// SIMATIC S7-200 project (STEP 7-Micro/WIN), CPU 224 REL 02.01

SYMBOL_TABLE USER1
S0               I0.0     // EMERGENCY pushbutton for the control unit
S1               I0.1     // START green pushbutton for the control unit
S2               I0.2     // STOP red pushbutton for the control unit
S3               I0.3     // START green pushbutton for the control unit
S4               I0.4     // STOP red pushbutton for the control unit
S5               I0.5     // Inductive sensor for the conveyor unit 2
S6               I0.6     // Capacitive sensor for the conveyor unit 2
S11              I1.1     // Capacitive sensor for the conveyor unit 1
S12              I1.2     // REED limit switch for the conveyor unit 1
S13              I1.3     // REED limit switch for the conveyor unit 1
S14              I1.4     // REED limit switch for the conveyor unit 1
S3_OFF           M0.0     // Memory to turn off latch attached to S3
SS3              M0.1     // Output for latch attached to S3
R_T1             M0.2     // Internal relay to reset TIMER1
ALL_LAMP         M0.3     // Output to flash lamps H1, H2, H3 and H4
GREEN            M0.4     // Output to turn H1 and H3 permanently on for start run
S1_OFF           M0.5     // Memory to turn off latch attached to S1
SS1              M0.6     // Output for latch attached to S1
STOP_K2          M0.7     // Contact to stop K2 when piece is detected after 2 seconds
S13_OFF          M1.0     // Memory to turn off latch attached to S13
SS13_K1          M1.1     // Output for latch attached to S13 to start motor K1
SS13_K2          M1.2     // Output to start motor K2 when the pick and place unit is returning
SS5              M1.3     // Output for latch S6 the capacitive sensor
SS6              M1.4     // Output for latch S6 the capacitive sensor
C_STOP_K1        M1.5     // Stop conveyor belt 2 some time after capacitive piece is sensed
I_STOP_K1        M1.6     // Stop conveyor belt 2 some time after inductive piece is sensed
E_STOP           M1.7     // Activates EMERGENCY situation
S_STOP           M2.0     // Activates STOP situation
SS11             M2.1     // Latch for S11
S_STOP_OFF       M2.2     // Exit STOP Situation
E_STOP_OFF       M2.3     // Exit EMERGENCY Situation
RED              M2.4     // Output to stop flashing in emergency situation
S_H4             M2.5     // Output for lamp H4 in stop situation
Y8               Q0.0     // Solenoid valve for vacuum unit
H1               Q0.1     // Green Lamp pushbutton for the control unit
H2               Q0.2     // Red Lamp pushbutton for the control unit
H3               Q0.3     // Green Lamp pushbutton for the control unit
H4               Q0.4     // Red lamp pushbutton for the control unit
K1               Q1.0     // AC 1 phase motor relay for the conveyor unit 2
K2               Q1.1     // AC 1 phase motor relay for the conveyor unit 1
Y2               Q2.2     // Pushing cylinder solenoid valve for inuductive pieces
Y3               Q2.3     // Pushing cylinder solenoid valve for capacitive pieces
Y4               Q2.4     // Solenoid valve for magazine pieces pushing cylinder conveyor unit 1
Y5               Q2.5     // Solenoid valve for transport cylinder delivery conveyor unit 1
Y6               Q2.6     // Solenoid valve for transport cylinder return conveyour unit 1
Y7               Q2.7     // Solenoid valve for vacuum unit lifting cylinder conveyour unit 1
TIMER1           T37      // TON timer to flash all the lights
TIMER2           T38      // TON timer to check if piece is detected by S11
TIMER3           T39      // TON timer for events after a piece has been detected
TIMER4           T41      // TON timer started by inductive load being sensed
TIMER5           T42      // TON timer started by capacitive load being sensed
END_SYMBOL_TABLE

ORGANIZATION_BLOCK MAIN:OB1
TITLE=PROGRAM COMMENTS
BEGIN
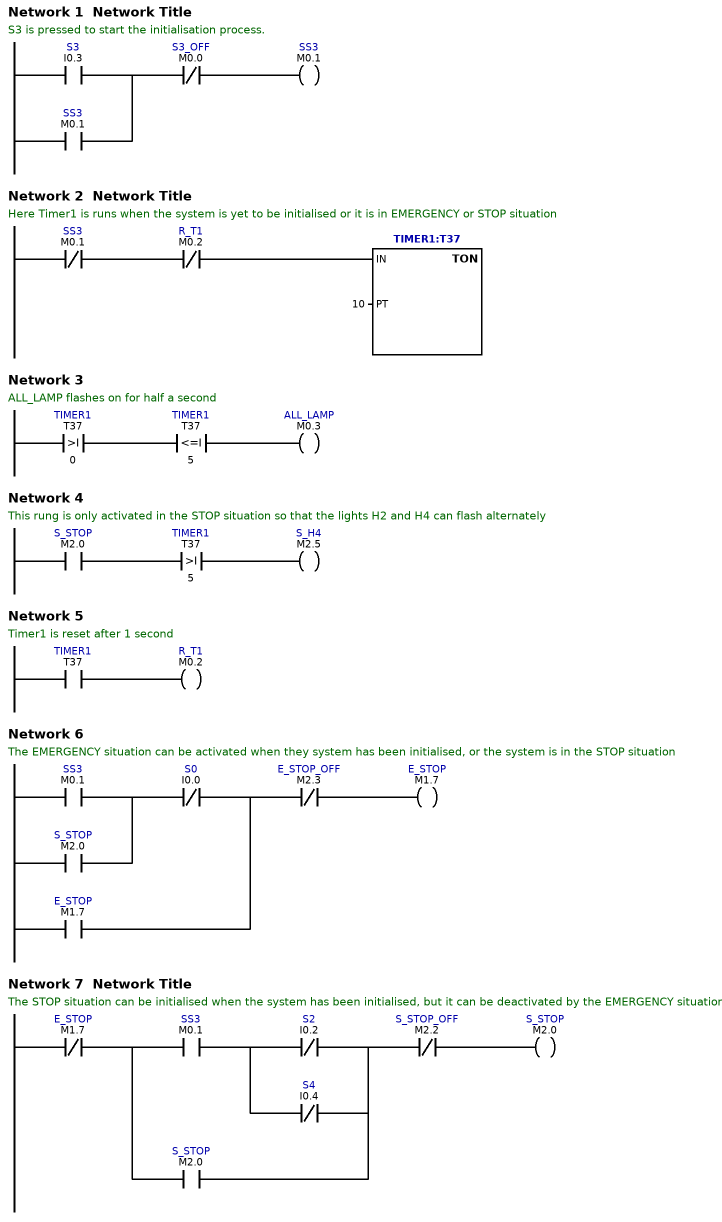
Network 1 // Network Title
// S3 is pressed to start the initialisation process.
LD     S3:I0.3
O      SS3:M0.1
AN     S3_OFF:M0.0
=      SS3:M0.1
Network 2 // Network Title
// Here Timer1 is runs when the system is yet to be initialised or it is in EMERGENCY or STOP situation
LDN    SS3:M0.1
AN     R_T1:M0.2
TON    TIMER1:T37, 10
Network 3
// ALL_LAMP flashes on for half a second
LDW>   TIMER1:T37, 0
AW<=   TIMER1:T37, 5
=      ALL_LAMP:M0.3
Network 4
// This rung is only activated in the STOP situation so that the lights H2 and H4 can flash alternately
// (network saved uncompiled; LAD cells follow)
// row 0: c0 -| |- S_STOP:M2.0  c1 -|>I|- TIMER1:T37, 5  c2 -( ) S_H4:M2.5
Network 5
// Timer1 is reset after 1 second
LD     TIMER1:T37
=      R_T1:M0.2
Network 6
// The EMERGENCY situation can be activated when they system has been initialised, or the system is in the STOP situation
// (network saved uncompiled; LAD cells follow)
// row 0: c0 -| |- SS3:M0.1 v  c1 -|/|- S0:I0.0 v  c2 -|/|- E_STOP_OFF:M2.3  c3 -( ) E_STOP:M1.7
// row 1: c0 -| |- S_STOP:M2.0 ^  c1 ^v
// row 2: c0 -| |- E_STOP:M1.7  c1 -- ^
Network 7 // Network Title
// The STOP situation can be initialised when the system has been initialised, but it can be deactivated by the EMERGENCY situation.
// (network saved uncompiled; LAD cells follow)
// row 0: c0 -|/|- E_STOP:M1.7 v  c1 -| |- SS3:M0.1 v  c2 -|/|- S2:I0.2 v  c3 -|/|- S_STOP_OFF:M2.2  c4 -( ) S_STOP:M2.0
// row 1: c0 ^v  c1 ^  c2 -|/|- S4:I0.4 ^v
// row 2: c0 ^  c1 -| |- S_STOP:M2.0  c2 -- ^
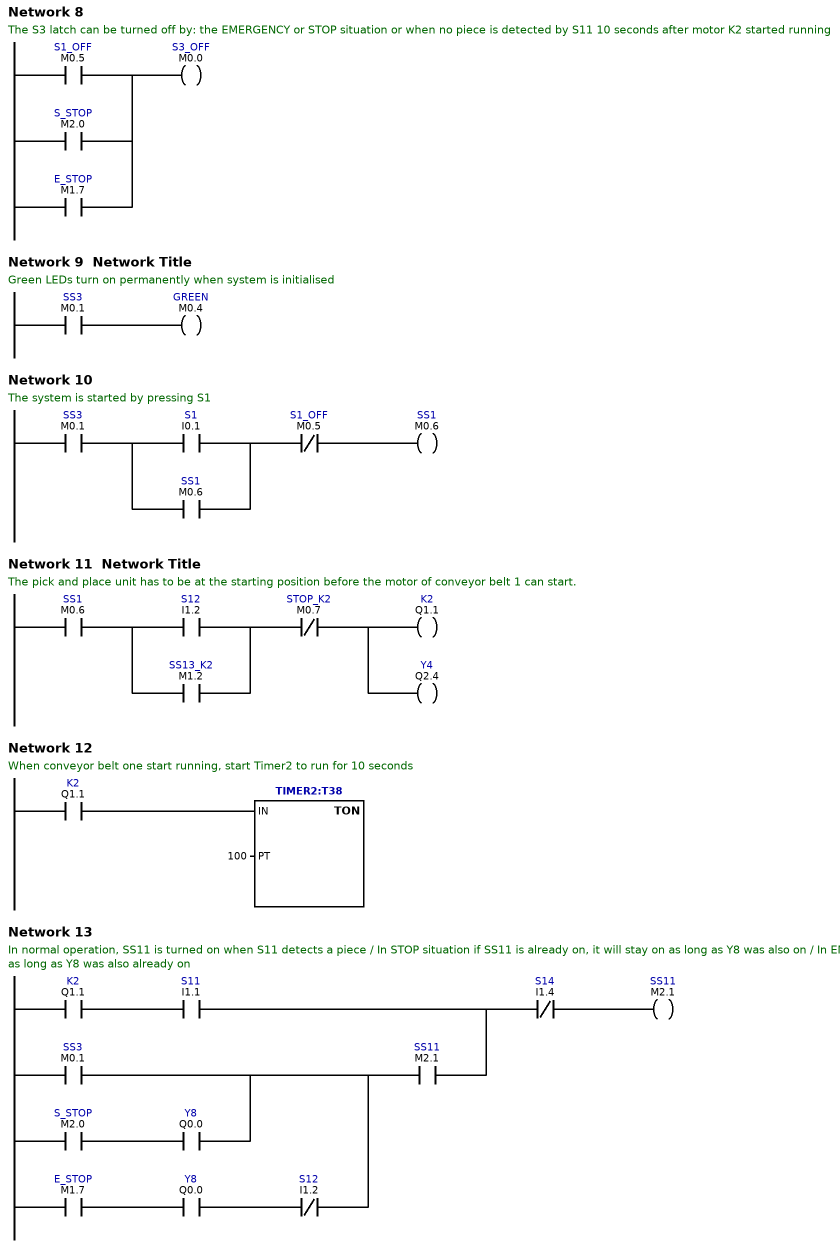
Network 8
// The S3 latch can be turned off by: the EMERGENCY or STOP situation or when no piece is detected by S11 10 seconds after motor K2 started running
// (network saved uncompiled; LAD cells follow)
// row 0: c0 -| |- S1_OFF:M0.5 v  c1 -( ) S3_OFF:M0.0
// row 1: c0 -| |- S_STOP:M2.0 ^v
// row 2: c0 -| |- E_STOP:M1.7 ^
Network 9 // Network Title
// Green LEDs turn on permanently when system is initialised
LD     SS3:M0.1
=      GREEN:M0.4
Network 10
// The system is started by pressing S1
LD     SS3:M0.1
LD     S1:I0.1
O      SS1:M0.6
ALD
AN     S1_OFF:M0.5
=      SS1:M0.6
Network 11 // Network Title
// The pick and place unit has to be at the starting position before the motor of conveyor belt 1 can start.
// (network saved uncompiled; LAD cells follow)
// row 0: c0 -| |- SS1:M0.6 v  c1 -| |- S12:I1.2 v  c2 -|/|- STOP_K2:M0.7 v  c3 -( ) K2:Q1.1
// row 1: c0 ^  c1 -| |- SS13_K2:M1.2 ^  c2 ^  c3 -( ) Y4:Q2.4
Network 12
// When conveyor belt one start running, start Timer2 to run for 10 seconds
LD     K2:Q1.1
TON    TIMER2:T38, 100
Network 13
// In normal operation, SS11 is turned on when S11 detects a piece
// In STOP situation if SS11 is already on, it will stay on as long as Y8 was also on
// In EMERGENCY if SS11 is already on, it will stay on as long as Y8 was also already on
// (network saved uncompiled; LAD cells follow)
// row 0: c0 -| |- K2:Q1.1  c1 -| |- S11:I1.1  c2 --  c3 -- v  c4 -|/|- S14:I1.4  c5 -( ) SS11:M2.1
// row 1: c0 -| |- SS3:M0.1  c1 -- v  c2 -- v  c3 -| |- SS11:M2.1 ^
// row 2: c0 -| |- S_STOP:M2.0  c1 -| |- Y8:Q0.0 ^  c2 ^v
// row 3: c0 -| |- E_STOP:M1.7  c1 -| |- Y8:Q0.0  c2 -|/|- S12:I1.2 ^
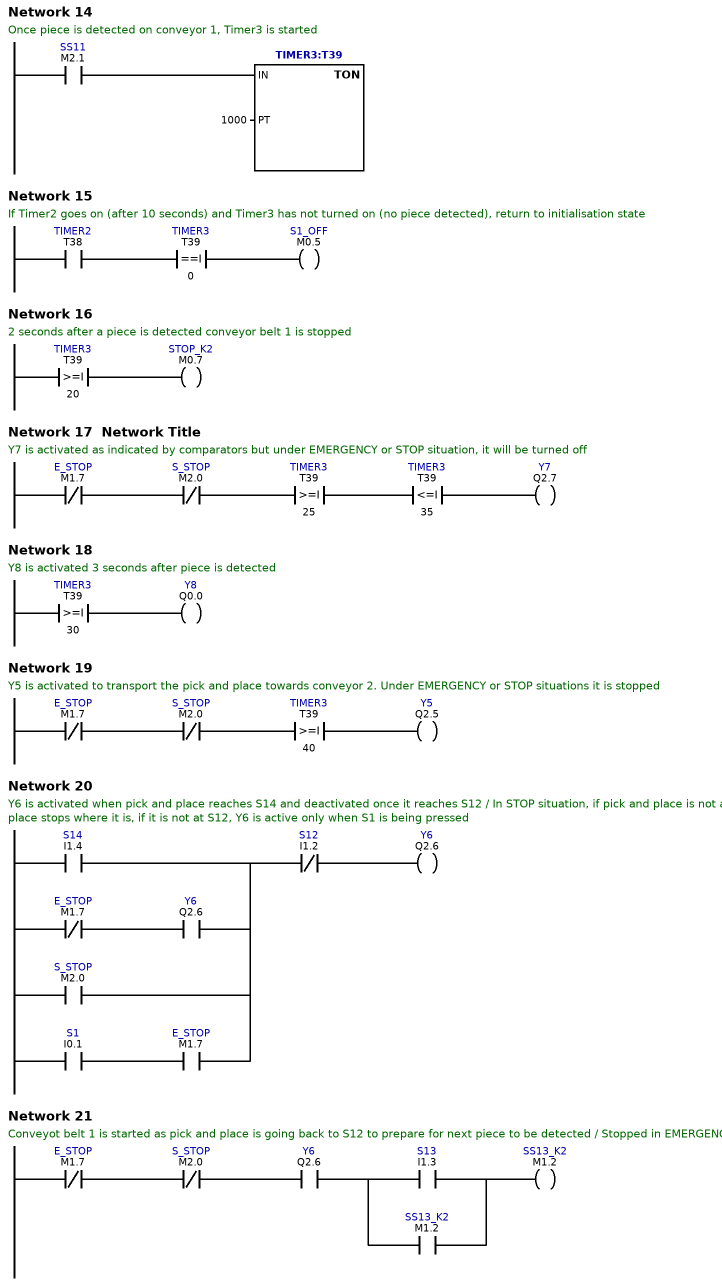
Network 14
// Once piece is detected on conveyor 1, Timer3 is started
// (network saved uncompiled; LAD cells follow)
// row 0: c0 -| |- SS11:M2.1  c1 --  c2 [TON TIMER3:T39 IN:=power@row0, PT:=1000]
// row 1: c2 [box]
Network 15
// If Timer2 goes on (after 10 seconds) and Timer3 has not turned on (no piece detected), return to initialisation state
LD     TIMER2:T38
AW=    TIMER3:T39, 0
=      S1_OFF:M0.5
Network 16
// 2 seconds after a piece is detected conveyor belt 1 is stopped
LDW>=  TIMER3:T39, 20
=      STOP_K2:M0.7
Network 17 // Network Title
// Y7 is activated as indicated by comparators but under EMERGENCY or STOP situation, it will be turned off
// (network saved uncompiled; LAD cells follow)
// row 0: c0 -|/|- E_STOP:M1.7  c1 -|/|- S_STOP:M2.0  c2 -|>=I|- TIMER3:T39, 25  c3 -|<=I|- TIMER3:T39, 35  c4 -( ) Y7:Q2.7
Network 18
// Y8 is activated 3 seconds after piece is detected
LDW>=  TIMER3:T39, 30
=      Y8:Q0.0
Network 19
// Y5 is activated to transport the pick and place towards conveyor 2. Under EMERGENCY or STOP situations it is stopped
// (network saved uncompiled; LAD cells follow)
// row 0: c0 -|/|- E_STOP:M1.7  c1 -|/|- S_STOP:M2.0  c2 -|>=I|- TIMER3:T39, 40  c3 -( ) Y5:Q2.5
Network 20
// Y6 is activated when pick and place reaches S14 and deactivated once it reaches S12
// In STOP situation, if pick and place is not at S12, Y6 is activated to return it
// In EMERGENCY situation, pick and place stops where it is, if it is not at S12, Y6 is active only when S1 is being pressed
// (network saved uncompiled; LAD cells follow)
// row 0: c0 -| |- S14:I1.4  c1 -- v  c2 -|/|- S12:I1.2  c3 -( ) Y6:Q2.6
// row 1: c0 -|/|- E_STOP:M1.7  c1 -| |- Y6:Q2.6 ^v
// row 2: c0 -| |- S_STOP:M2.0  c1 -- ^v
// row 3: c0 -| |- S1:I0.1  c1 -| |- E_STOP:M1.7 ^
Network 21
// Conveyot belt 1 is started as pick and place is going back to S12 to prepare for next piece to be detected
// Stopped in EMERGENCY and STOP situation
// (network saved uncompiled; LAD cells follow)
// row 0: c0 -|/|- E_STOP:M1.7  c1 -|/|- S_STOP:M2.0  c2 -| |- Y6:Q2.6 v  c3 -| |- S13:I1.3 v  c4 -( ) SS13_K2:M1.2
// row 1: c2 ^  c3 -| |- SS13_K2:M1.2 ^
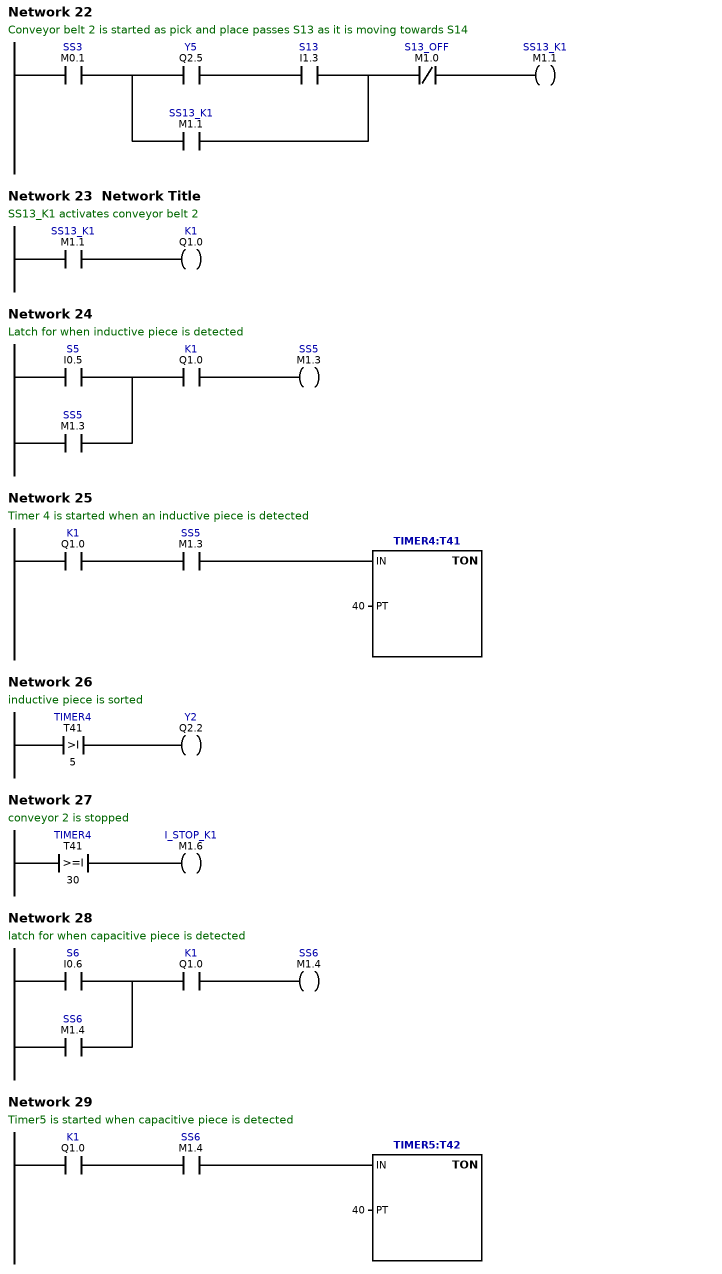
Network 22
// Conveyor belt 2 is started as pick and place passes S13 as it is moving towards S14
LD     SS3:M0.1
LD     Y5:Q2.5
A      S13:I1.3
O      SS13_K1:M1.1
ALD
AN     S13_OFF:M1.0
=      SS13_K1:M1.1
Network 23 // Network Title
// SS13_K1 activates conveyor belt 2
LD     SS13_K1:M1.1
=      K1:Q1.0
Network 24
// Latch for when inductive piece is detected
// (network saved uncompiled; LAD cells follow)
// row 0: c0 -| |- S5:I0.5 v  c1 -| |- K1:Q1.0  c2 -( ) SS5:M1.3
// row 1: c0 -| |- SS5:M1.3 ^
Network 25
// Timer 4 is started when an inductive piece is detected
// (network saved uncompiled; LAD cells follow)
// row 0: c0 -| |- K1:Q1.0  c1 -| |- SS5:M1.3  c2 --  c3 [TON TIMER4:T41 IN:=power@row0, PT:=40]
// row 1: c3 [box]
Network 26
// inductive piece is sorted
LDW>   TIMER4:T41, 5
=      Y2:Q2.2
Network 27
// conveyor 2 is stopped
// (network saved uncompiled; LAD cells follow)
// row 0: c0 -|>=I|- TIMER4:T41, 30  c1 -( ) I_STOP_K1:M1.6
Network 28
// latch for when capacitive piece is detected
// (network saved uncompiled; LAD cells follow)
// row 0: c0 -| |- S6:I0.6 v  c1 -| |- K1:Q1.0  c2 -( ) SS6:M1.4
// row 1: c0 -| |- SS6:M1.4 ^
Network 29
// Timer5 is started when capacitive piece is detected
// (network saved uncompiled; LAD cells follow)
// row 0: c0 -| |- K1:Q1.0  c1 -| |- SS6:M1.4  c2 --  c3 [TON TIMER5:T42 IN:=power@row0, PT:=40]
// row 1: c3 [box]
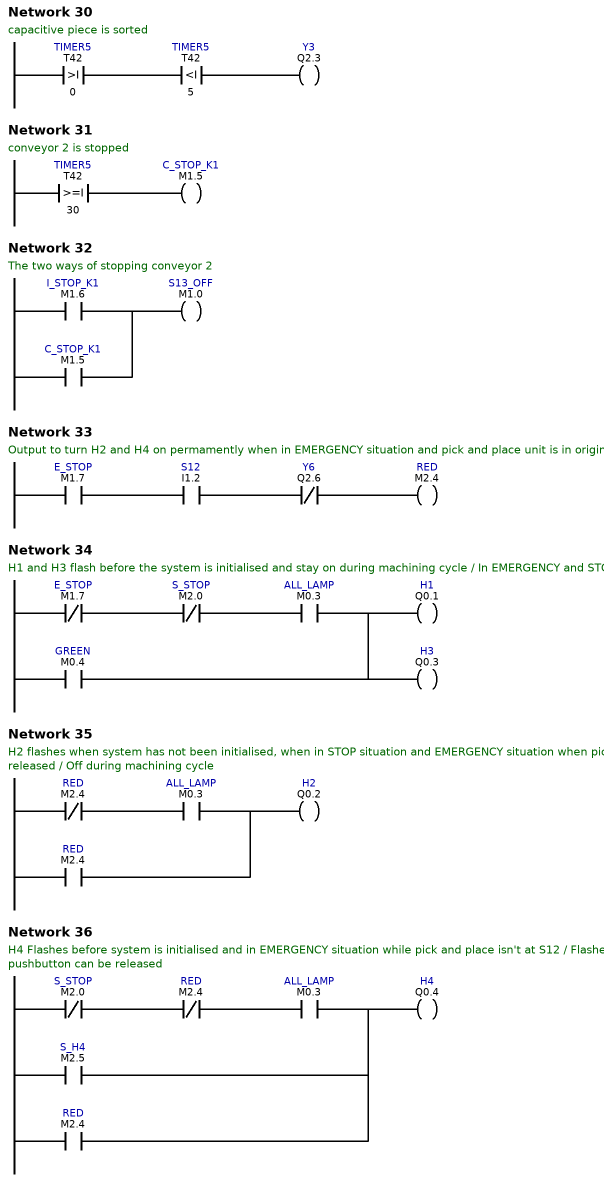
Network 30
// capacitive piece is sorted
LDW>   TIMER5:T42, 0
AW<    TIMER5:T42, 5
=      Y3:Q2.3
Network 31
// conveyor 2 is stopped
// (network saved uncompiled; LAD cells follow)
// row 0: c0 -|>=I|- TIMER5:T42, 30  c1 -( ) C_STOP_K1:M1.5
Network 32
// The two ways of stopping conveyor 2
// (network saved uncompiled; LAD cells follow)
// row 0: c0 -| |- I_STOP_K1:M1.6 v  c1 -( ) S13_OFF:M1.0
// row 1: c0 -| |- C_STOP_K1:M1.5 ^
Network 33
// Output to turn H2 and H4 on permamently when in EMERGENCY situation and pick and place unit is in original position. This is to show that the EMERGENCY button can be released
// (network saved uncompiled; LAD cells follow)
// row 0: c0 -| |- E_STOP:M1.7  c1 -| |- S12:I1.2  c2 -|/|- Y6:Q2.6  c3 -( ) RED:M2.4
Network 34
// H1 and H3 flash before the system is initialised and stay on during machining cycle
// In EMERGENCY and STOP situation they are off
// (network saved uncompiled; LAD cells follow)
// row 0: c0 -|/|- E_STOP:M1.7  c1 -|/|- S_STOP:M2.0  c2 -| |- ALL_LAMP:M0.3 v  c3 -( ) H1:Q0.1
// row 1: c0 -| |- GREEN:M0.4  c1 --  c2 -- ^  c3 -( ) H3:Q0.3
Network 35
// H2 flashes when system has not been initialised, when in STOP situation and EMERGENCY situation when pick and place unit is not at original location.
// It stays on when EMERGENCY button can be released
// Off during machining cycle
// (network saved uncompiled; LAD cells follow)
// row 0: c0 -|/|- RED:M2.4  c1 -| |- ALL_LAMP:M0.3 v  c2 -( ) H2:Q0.2
// row 1: c0 -| |- RED:M2.4  c1 -- ^
Network 36
// H4 Flashes before system is initialised and in EMERGENCY situation while pick and place isn't at S12
// Flashes alternately to H2 when in STOP situation
// Stays on in EMERGENCY situation when the pushbutton can be released
// (network saved uncompiled; LAD cells follow)
// row 0: c0 -|/|- S_STOP:M2.0  c1 -|/|- RED:M2.4  c2 -| |- ALL_LAMP:M0.3 v  c3 -( ) H4:Q0.4
// row 1: c0 -| |- S_H4:M2.5  c1 --  c2 -- ^v
// row 2: c0 -| |- RED:M2.4  c1 --  c2 -- ^
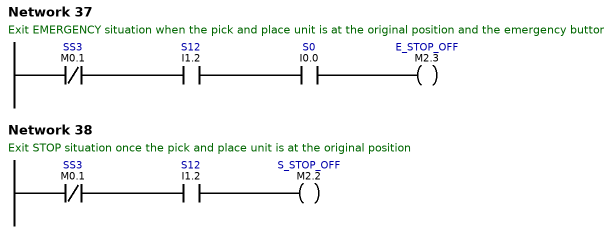
Network 37
// Exit EMERGENCY situation when the pick and place unit is at the original position and the emergency button is released
// (network saved uncompiled; LAD cells follow)
// row 0: c0 -|/|- SS3:M0.1  c1 -| |- S12:I1.2  c2 -| |- S0:I0.0  c3 -( ) E_STOP_OFF:M2.3
Network 38
// Exit STOP situation once the pick and place unit is at the original position
// (network saved uncompiled; LAD cells follow)
// row 0: c0 -|/|- SS3:M0.1  c1 -| |- S12:I1.2  c2 -( ) S_STOP_OFF:M2.2
END_ORGANIZATION_BLOCK
